Fanuc KAREL source: kt00293.compact.KL

PROGRAM KT00293
%STACKSIZE=65535
%PRIORITY=65535
%NOLOCKGROUP
VAR
I1 : INTEGER
I2 : INTEGER
OUT : BOOLEAN
BEGIN
I1=2
I2=3
I1=2
I2=3
OUT=(I1 <> I2)
END KT00293
